{attribute 'qualified_only'}
VAR_GLOBAL CONSTANT
  //-----------------------------------------------------------------------------
  // file paths for message system
  //  - compiler define option WIN switches to Windows file paths
  //-----------------------------------------------------------------------------
{IF NOT defined (BSD)}
  {info 'PLC_MOTION_LAYER: WIN'}
  LOG_DIR               : STRING  := 'C:\TwinCAT\#MsgFiles\';
{ELSE}
  {info 'PLC_MOTION_LAYER: BSD'}
  LOG_DIR               : STRING  := '/usr/local/etc/TwinCAT/#MsgFiles/';
{END_IF}

  LOG_FILE              : STRING  := 'MSG_EXT_';

  MAX_MESSAGE           : UINT     := 200; // max entry in message list
END_VAR
VAR_GLOBAL
  fbLocalTime                     : fb_LocalTime;
  dtLocalTime                     : DT;
  sLocalTime                      : STRING;

  Messages                        : ARRAY[1..MAX_MESSAGE] OF ST_Message;
  MessageIndex                    : UINT := 0; // message index
  MessageError                    : UINT := 0; // error counter

  MessageLevelAxisPtp             : E_MessageType := E_MessageType.eMessageError;
  MessageLevelAxisCam             : E_MessageType := E_MessageType.eMessageError;
  MessageLevelNciChn              : E_MessageType := E_MessageType.eMessageError;

  MessageLevelTriggerBox          : ARRAY[1..PLC_CONSTANT.MAX_TRIGGER_BOX]  OF E_MessageType;
  MessageLevelTouchProbe          : ARRAY[1..PLC_CONSTANT.MAX_TOUCH_PROBE]  OF E_MessageType;

END_VAR

(* stored: Version 1.1.0.1
   GVL GVL_MSG: Id {74e20592-95e1-442c-8a34-d2e8b89ee769} *)
